FUNCTION_BLOCK FB_Skill_1 EXTENDS FB_Base IMPLEMENTS  ITF_1_Skill
VAR_INPUT
	SFCInit, SFCPause, SFCReset: BOOL;
END_VAR
VAR_OUTPUT
	bBusy, bDone: BOOL;
	SFCError: BOOL;
	SFCCurrentStep: STRING;
END_VAR
VAR
	SubSkillHandler : FB_SkillHandler;
END_VAR

{warning 'Add method implementation '}
METHOD M_Pause : BOOL
IF _state=eState.Active THEN
	SFCPause:=TRUE;
END_IF
END_METHOD

{warning 'Add method implementation '}
METHOD M_Restart : BOOL //Stay activ, but restart
SFCReset:=True;
END_METHOD

{warning 'Add method implementation '}
METHOD M_Resume : BOOL
SFCPause:=False;
END_METHOD

{warning 'Add method implementation '}
METHOD M_Start : BOOL
Activate();
END_METHOD

{warning 'Add method implementation '}
METHOD M_Stop : BOOL
IF _state=eState.Active THEN
	SFCPause:=TRUE;
	super^.Deactivate();
END_IF
END_METHOD

METHOD onActivate : BOOL
// ---- Init ----
transitionresult:=eResult.None;



// ---- Change ----




// ---- Check ----
transitionresult := eResult.SUCCESS;


// ---- Change State ----
IF transitionresult= eResult.SUCCESS THEN
	State:=eState.Active;
ELSIF transitionresult= eResult.FAILURE THEN
	State:=eState.Inactive;
ELSIF transitionresult= eResult.ERROR THEN
	State:=eState.ErrorProcessing;
ELSE
	ADSLOGSTR(ADSLOG_MSGTYPE_WARN,'Transitionresult from onActivate is None','');
END_IF
END_METHOD

METHOD onCleanup : BOOL
// ---- Init ----
transitionresult:=eResult.None;



// ---- Change ----



// ---- Check ----
transitionresult := eResult.SUCCESS;


// ---- Change State ----
IF transitionresult= eResult.SUCCESS THEN
	State:=eState.Unconfigured;
ELSIF transitionresult= eResult.FAILURE THEN
	ADSLOGSTR(ADSLOG_MSGTYPE_WARN,'Transitionresult from onCleanup is FAILURE ','');
ELSIF transitionresult= eResult.ERROR THEN
	State:=eState.ErrorProcessing;
ELSE
	ADSLOGSTR(ADSLOG_MSGTYPE_WARN,'Transitionresult from onCleanup is NONE','');
END_IF
END_METHOD

METHOD onConfigure : BOOL
// ---- Init ----
transitionresult:=eResult.None;



// ---- Change ----


// ---- Check ----
transitionresult := eResult.SUCCESS;


// ---- Change State ----
IF transitionresult= eResult.SUCCESS THEN
	State:=eState.Inactive;
ELSIF transitionresult= eResult.FAILURE THEN
	State:=eState.Unconfigured;
ELSIF transitionresult= eResult.ERROR THEN
	State:=eState.ErrorProcessing;
ELSE
	ADSLOGSTR(ADSLOG_MSGTYPE_WARN,'Transitionresult from onConfigure is None','');
END_IF
END_METHOD

METHOD onDeactivate : BOOL
// ---- Init ----
transitionresult:=eResult.None;



// ---- Change ----
 //Stopping SFC



// ---- Check ----
transitionresult := eResult.SUCCESS;


// ---- Change State ----
IF transitionresult= eResult.SUCCESS THEN
	State:=eState.Inactive;
ELSIF transitionresult= eResult.FAILURE THEN
	ADSLOGSTR(ADSLOG_MSGTYPE_WARN,'Transitionresult from onDeactivate is FAILURE','');
ELSIF transitionresult= eResult.ERROR THEN
	State:=eState.ErrorProcessing;
ELSE
	ADSLOGSTR(ADSLOG_MSGTYPE_WARN,'Transitionresult from onDeactivate is None','');
END_IF
END_METHOD

METHOD onError : BOOL
// ---- Init ----
transitionresult:=eResult.None;



// ---- Change ----





// ---- Check ----
transitionresult := eResult.SUCCESS;


// ---- Change State ----
IF transitionresult= eResult.SUCCESS THEN
	State:=eState.Unconfigured;
ELSIF transitionresult= eResult.FAILURE THEN
	State:=eState.Finalized;
ELSIF transitionresult= eResult.ERROR THEN
	ADSLOGSTR(ADSLOG_MSGTYPE_WARN,'Transitionresult from onError is Error','');
ELSE
	ADSLOGSTR(ADSLOG_MSGTYPE_WARN,'Transitionresult from onError is None','');
END_IF
END_METHOD

METHOD onShutdown : BOOL
// ---- Init ----
transitionresult:=eResult.None;



// ---- Change ----




// ---- Check ----
transitionresult := eResult.SUCCESS;


// ---- Change State ----
IF transitionresult= eResult.SUCCESS THEN
	State:=eState.Finalized;
ELSIF transitionresult= eResult.FAILURE THEN
	ADSLOGSTR(ADSLOG_MSGTYPE_WARN,'Transitionresult from onShutdown is FAILURE','');
ELSIF transitionresult= eResult.ERROR THEN
	State:=eState.ErrorProcessing;
ELSE
	ADSLOGSTR(ADSLOG_MSGTYPE_WARN,'Transitionresult from onShutdown is None','');
END_IF
END_METHOD

{warning 'Add property implementation'}
PROPERTY P_Busy : BOOL
GET
IF _state=eState.Active THEN
	P_Busy:=TRUE;
ELSE
	P_Busy:=FALSE;
END_IF
END_GET
END_PROPERTY

{warning 'Add property implementation'}
PROPERTY P_Done : BOOL
GET
P_Done:=bDone;
END_GET
END_PROPERTY

END_FUNCTION_BLOCK

(* stored: Version 1.1.0.1, ProductVersion 3.1.4026.18
   POU FB_Skill_1: Id {a3adf140-2c5e-4b25-b32d-7f3481940825}, SpecialFunc None
   Folder StateControl: Id {a37ba031-65ef-4b21-b6e0-5be6b4f114a7}
   Method M_Pause: Id {a0cc9d07-14cd-42d7-b54a-a5fbf50b866e}
   Method M_Restart: Id {66dafe8b-cff0-4d6c-b567-3cd4c76f83e6}
   Method M_Resume: Id {90162248-4a73-47ab-a686-27f06d6359f8}
   Method M_Start: Id {8bec1e83-9088-4ef4-8c5a-f447585bacf1}
   Method M_Stop: Id {e1ac8d39-e526-43c9-aa2e-b224c81d49dd}
   Method onActivate: Id {2a45bebb-20de-4d79-9c69-ff3636c276d5}
   Method onCleanup: Id {a9025233-87bf-467b-af88-11c81eabb531}
   Method onConfigure: Id {40239a8d-224a-404f-bf74-2f20a267433a}
   Method onDeactivate: Id {73886f48-defb-4d50-b015-62459c93f7ac}
   Method onError: Id {5e6ed6d0-486d-4b72-99d4-f75ac8596220}
   Method onShutdown: Id {d749c111-3627-44d4-89d2-aa63e97b3dd3}
   Property P_Busy: Id {291a7649-1bc4-455f-a684-4385fb95268c}
   Get Get: Id {43aba8cd-02e2-49d3-a8d0-2861f457d08c}
   Property P_Done: Id {acf7213a-745b-4834-b565-bde144be80a9}
   Get Get: Id {70e1d4e4-4783-4e1a-b0aa-d54aa022259a} *)
